FUNCTION_BLOCK INTERNAL fbTaskTests EXTENDS fbComponent
VAR			
	_task_index : UINT;
	_tasks : ARRAY[0..NUMBER_OF_TASKS] OF fbTask(THIS^); 
	_task_lock_group : ARRAY[0..NUMBER_OF_TASKS] OF UINT;
	_task_done_condition : ARRAY[0..NUMBER_OF_TASKS] OF BOOL;	
	_task_fail_condition : ARRAY[0..NUMBER_OF_TASKS] OF BOOL; 	
END_VAR

VAR CONSTANT
	NUMBER_OF_TASKS : UINT := 4;
END_VAR

_task_index := 0;
IF(_tasks[_task_index].Execute(_task_lock_group[_task_index])) THEN
	_tasks[_task_index].DoneWhen(_task_done_condition[_task_index]);
	_tasks[_task_index].ThrowWhen(_task_fail_condition[_task_index]);
END_IF


_task_index := _task_index + 1;
IF(_tasks[_task_index].Execute(_task_lock_group[_task_index])) THEN
	_tasks[_task_index].DoneWhen(_task_done_condition[_task_index]);
	_tasks[_task_index].ThrowWhen(_task_fail_condition[_task_index]);
END_IF

_task_index := _task_index + 1;
IF(_tasks[_task_index].Execute(_task_lock_group[_task_index])) THEN
	_tasks[_task_index].DoneWhen(_task_done_condition[_task_index]);
	_tasks[_task_index].ThrowWhen(_task_fail_condition[_task_index]);
END_IF

_task_index := _task_index + 1;
IF(_tasks[_task_index].Execute(_task_lock_group[_task_index])) THEN
	_tasks[_task_index].DoneWhen(_task_done_condition[_task_index]);
	_tasks[_task_index].ThrowWhen(_task_fail_condition[_task_index]);
END_IF

_task_index := _task_index + 1;
IF(_tasks[_task_index].Execute(_task_lock_group[_task_index])) THEN
	_tasks[_task_index].DoneWhen(_task_done_condition[_task_index]);
	_tasks[_task_index].ThrowWhen(_task_fail_condition[_task_index]);
END_IF

{attribute 'TcRpcEnable'}
METHOD AbortTest
VAR_INPUT
	taskIndex : UINT;
END_VAR
THIS^._tasks[taskIndex].Reset();
END_METHOD

{attribute 'TcRpcEnable'}
METHOD GetBusyTest : BOOL;
VAR_INPUT
	taskIndex : UINT;
END_VAR
GetBusyTest := THIS^._tasks[taskIndex].Busy;
END_METHOD

{attribute 'TcRpcEnable'}
METHOD GetDoneTest : BOOL;
VAR_INPUT
	taskIndex : UINT;
END_VAR
GetDoneTest := THIS^._tasks[taskIndex].Done;
END_METHOD

{attribute 'TcRpcEnable'}
METHOD GetErrorTest : BOOL;
VAR_INPUT
	taskIndex : UINT;
END_VAR
GetErrorTest := THIS^._tasks[taskIndex].Error;
END_METHOD

METHOD InvokeTask : ITaskStatus
VAR_INPUT
	taskIndex : UINT;
END_VAR
THIS^._tasks[taskIndex].Invoke();
InvokeTask := THIS^._tasks[taskIndex];
END_METHOD

{attribute 'TcRpcEnable'}
METHOD InvokeTaskTest
VAR_INPUT
	taskIndex : UINT;
END_VAR
InvokeTask(taskIndex);
END_METHOD

{attribute 'TcRpcEnable'}
METHOD INTERNAL InvokeTaskTests_with_done : BOOL
VAR_INPUT
	taskIndex : UINT;
END_VAR
InvokeTaskTests_with_done := InvokeTask(taskIndex).Done;
END_METHOD

METHOD PROTECTED  ManualControl
END_METHOD

{attribute 'TcRpcEnable'}
METHOD ResetComponent
VAR_INPUT
END_VAR
THIS^.Lock := 0;
END_METHOD

{attribute 'TcRpcEnable'}
METHOD ResetTask
VAR_INPUT
	taskIndex : UINT;
END_VAR
THIS^._tasks[taskIndex].Reset();
END_METHOD

END_FUNCTION_BLOCK

(* stored: Version 1.1.0.1, ProductVersion 3.1.4024.5
   POU fbTaskTests: Id {a16465a5-946d-4b35-8086-ed37ba24b1a6}, SpecialFunc None
   Folder tests: Id {5613e13c-336e-4006-bf2b-04853f5c1b8c}
   Method AbortTest: Id {01635d81-a339-4f63-b04f-fc70f4821b30}
   Method GetBusyTest: Id {1c9c4af6-7170-4e64-8cd6-b2e233bd0762}
   Method GetDoneTest: Id {d11d4342-3b60-4195-b764-2b40f7d485c7}
   Method GetErrorTest: Id {a30dda01-48b0-4614-9f64-c034c3bf354d}
   Method InvokeTask: Id {4de76c8f-d566-4f35-b3c1-8f71883427b8}
   Method InvokeTaskTest: Id {d1efa48f-d85b-43b4-9493-511717509295}
   Method InvokeTaskTests_with_done: Id {7d366e2f-91aa-40ea-8d83-3190f7006b23}
   Method ManualControl: Id {8d20f903-74a6-4e83-891d-914170f40249}
   Method ResetComponent: Id {ae7b6d78-2fd1-47fe-bfc1-401d4f5d519a}
   Method ResetTask: Id {e2d6ab32-afce-4087-9c2e-1f46ce3d408d} *)
